PROGRAM MAIN
VAR
	bBlinker	: BOOL;
	tonBlink	: TON;
	sTime :TIME:= T#1S;
END_VAR


tonBlink(IN := NOT tonBlink.Q, PT := sTime);

IF tonBlink.Q THEN
	bBlinker := NOT bBlinker;
END_IF

END_PROGRAM

(* stored: Version 1.1.0.1, ProductVersion 3.1.4026.18
   POU MAIN: Id {ce6f4c4f-7373-443d-941b-4dfa87132aee}, SpecialFunc None *)
